// Mitsubishi GX Works2 project: REAL_PROJECT   PLC: Q03UDV

PROGRAM Manual
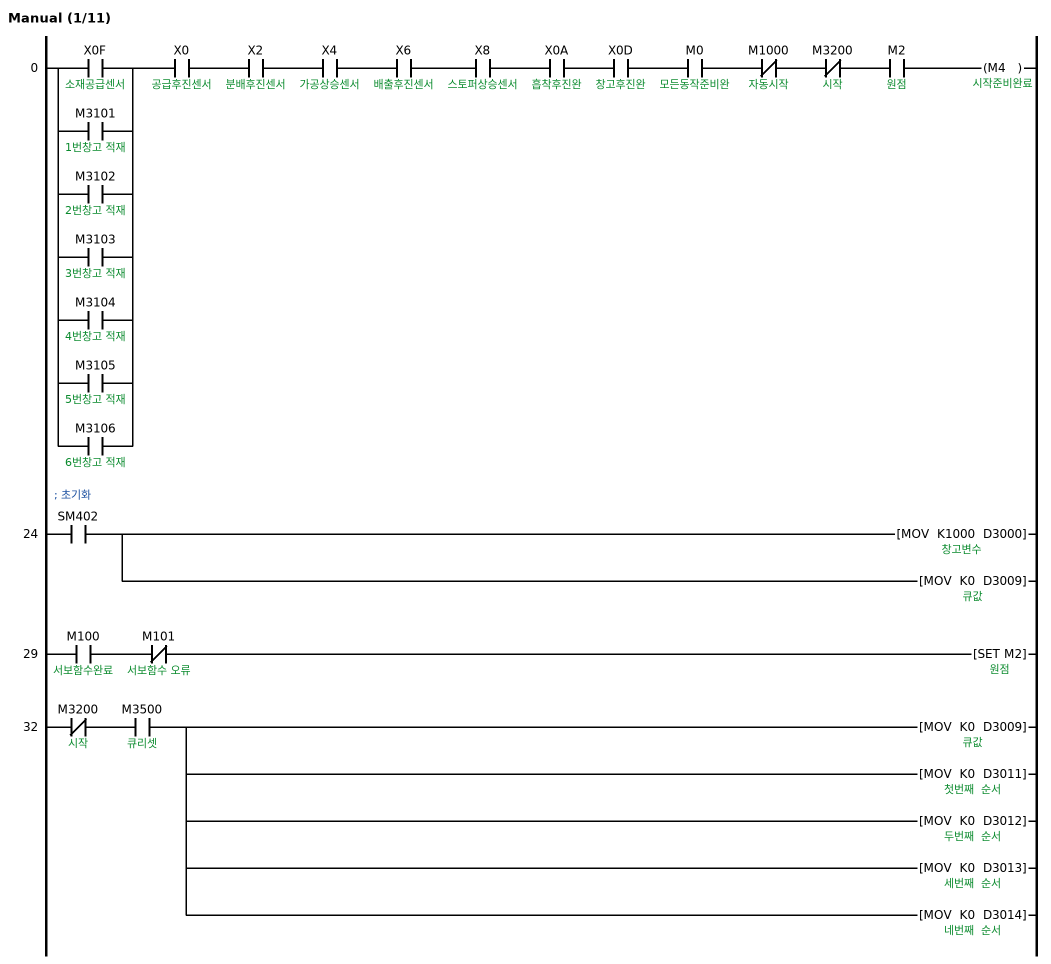
0     LD      X0F  ; 소재공급센서
      OR      M3101  ; 1번창고 적재
      OR      M3102  ; 2번창고 적재
      OR      M3103  ; 3번창고 적재
      OR      M3104  ; 4번창고 적재
      OR      M3105  ; 5번창고 적재
      OR      M3106  ; 6번창고 적재
      AND     X0  ; 공급후진센서
      AND     X2  ; 분배후진센서
      AND     X4  ; 가공상승센서
      AND     X6  ; 배출후진센서
      AND     X8  ; 스토퍼상승센서
      AND     X0A  ; 흡착후진완
      AND     X0D  ; 창고후진완
      AND     M0  ; 모든동작준비완
      ANI     M1000  ; 자동시작
      ANI     M3200  ; 시작
      AND     M2  ; 원점
      OUT     M4  ; 시작준비완료
; 초기화
24    LD      SM402
      MOV     K1000 D3000  ; 창고변수
      MOV     K0 D3009  ; 큐값
29    LD      M100  ; 서보함수완료
      ANI     M101  ; 서보함수 오류
      SET     M2  ; 원점
32    LDI     M3200  ; 시작
      AND     M3500  ; 큐리셋
      MOV     K0 D3009
      MOV     K0 D3011  ; 첫번째  순서
      MOV     K0 D3012  ; 두번째  순서
      MOV     K0 D3013  ; 세번째  순서
      MOV     K0 D3014  ; 네번째  순서
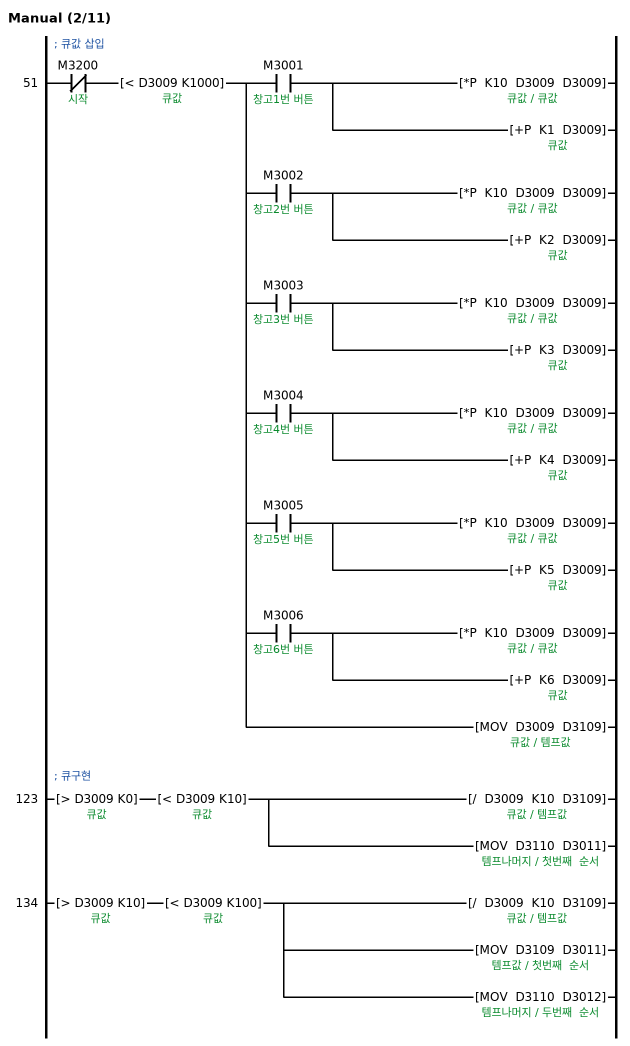
; 큐값 삽입
51    LDI     M3200  ; 시작
      AND<    D3009 K1000  ; 큐값
      MPS
      AND     M3001  ; 창고1번 버튼
      *P      K10 D3009 D3009
      +P      K1 D3009
      MRD
      AND     M3002  ; 창고2번 버튼
      *P      K10 D3009 D3009
      +P      K2 D3009
      MRD
      AND     M3003  ; 창고3번 버튼
      *P      K10 D3009 D3009
      +P      K3 D3009
      MRD
      AND     M3004  ; 창고4번 버튼
      *P      K10 D3009 D3009
      +P      K4 D3009
      MRD
      AND     M3005  ; 창고5번 버튼
      *P      K10 D3009 D3009
      +P      K5 D3009
      MRD
      AND     M3006  ; 창고6번 버튼
      *P      K10 D3009 D3009
      +P      K6 D3009
      MPP
      MOV     D3009 D3109  ; 템프값
; 큐구현
123   LD>     D3009 K0  ; 큐값
      AND<    D3009 K10  ; 큐값
      /       D3009 K10 D3109
      MOV     D3110 D3011  ; 템프나머지
134   LD>     D3009 K10  ; 큐값
      AND<    D3009 K100  ; 큐값
      /       D3009 K10 D3109
      MOV     D3109 D3011
      MOV     D3110 D3012
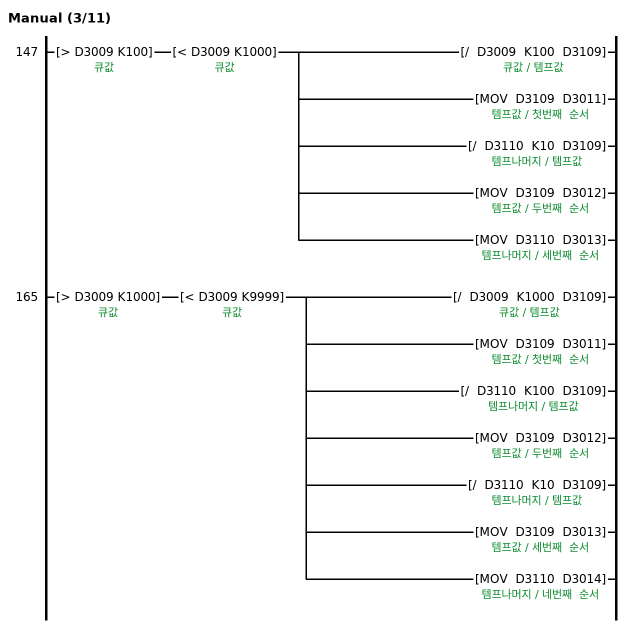
147   LD>     D3009 K100  ; 큐값
      AND<    D3009 K1000  ; 큐값
      /       D3009 K100 D3109
      MOV     D3109 D3011
      /       D3110 K10 D3109
      MOV     D3109 D3012
      MOV     D3110 D3013
165   LD>     D3009 K1000  ; 큐값
      AND<    D3009 K9999  ; 큐값
      /       D3009 K1000 D3109
      MOV     D3109 D3011
      /       D3110 K100 D3109
      MOV     D3109 D3012
      /       D3110 K10 D3109
      MOV     D3109 D3013
      MOV     D3110 D3014
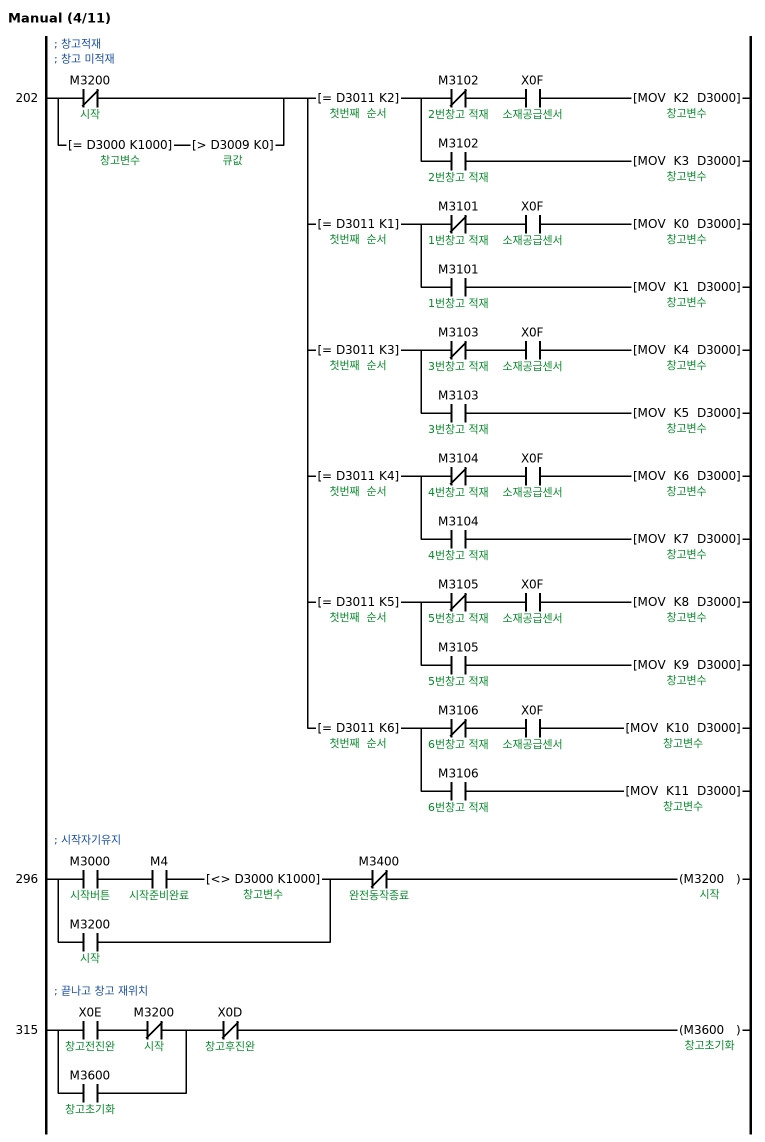
; 창고적재
; 창고 미적재
202   LDI     M3200  ; 시작
      LD=     D3000 K1000  ; 창고변수
      AND>    D3009 K0  ; 큐값
      ORB
      MPS
      AND=    D3011 K2  ; 첫번째  순서
      MPS
      ANI     M3102  ; 2번창고 적재
      AND     X0F  ; 소재공급센서
      MOV     K2 D3000
      MPP
      AND     M3102  ; 2번창고 적재
      MOV     K3 D3000
      MRD
      AND=    D3011 K1  ; 첫번째  순서
      MPS
      ANI     M3101  ; 1번창고 적재
      AND     X0F  ; 소재공급센서
      MOV     K0 D3000
      MPP
      AND     M3101  ; 1번창고 적재
      MOV     K1 D3000
      MRD
      AND=    D3011 K3  ; 첫번째  순서
      MPS
      ANI     M3103  ; 3번창고 적재
      AND     X0F  ; 소재공급센서
      MOV     K4 D3000
      MPP
      AND     M3103  ; 3번창고 적재
      MOV     K5 D3000
      MRD
      AND=    D3011 K4  ; 첫번째  순서
      MPS
      ANI     M3104  ; 4번창고 적재
      AND     X0F  ; 소재공급센서
      MOV     K6 D3000
      MPP
      AND     M3104  ; 4번창고 적재
      MOV     K7 D3000
      MRD
      AND=    D3011 K5  ; 첫번째  순서
      MPS
      ANI     M3105  ; 5번창고 적재
      AND     X0F  ; 소재공급센서
      MOV     K8 D3000
      MPP
      AND     M3105  ; 5번창고 적재
      MOV     K9 D3000
      MPP
      AND=    D3011 K6  ; 첫번째  순서
      MPS
      ANI     M3106  ; 6번창고 적재
      AND     X0F  ; 소재공급센서
      MOV     K10 D3000
      MPP
      AND     M3106  ; 6번창고 적재
      MOV     K11 D3000
; 시작자기유지
296   LD      M3000  ; 시작버튼
      AND     M4  ; 시작준비완료
      AND<>   D3000 K1000  ; 창고변수
      OR      M3200  ; 시작
      ANI     M3400  ; 완전동작종료
      OUT     M3200  ; 시작
; 끝나고 창고 재위치
315   LD      X0E  ; 창고전진완
      ANI     M3200  ; 시작
      OR      M3600  ; 창고초기화
      ANI     X0D  ; 창고후진완
      OUT     M3600  ; 창고초기화
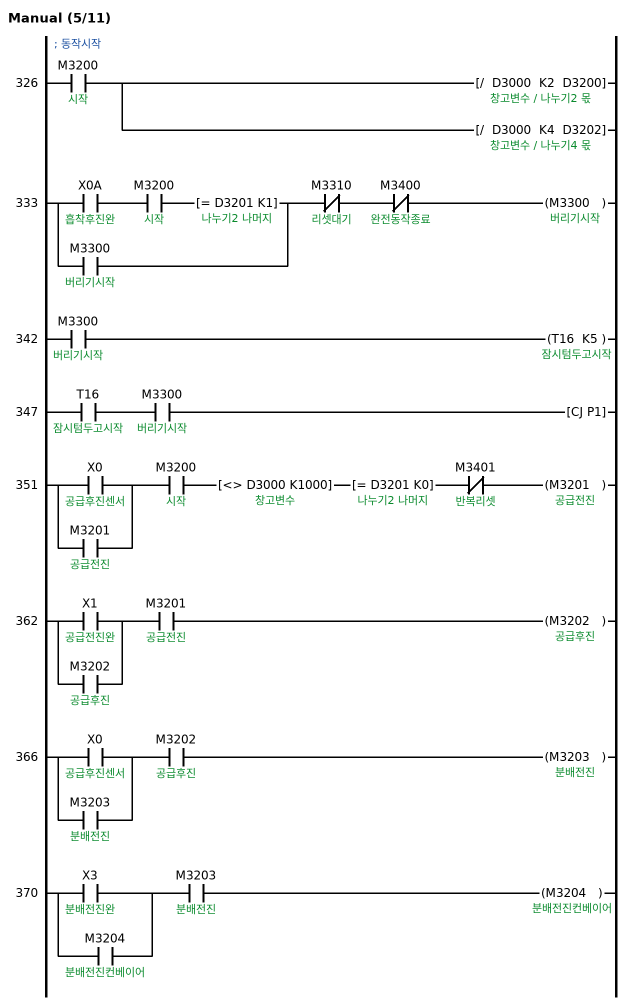
; 동작시작
326   LD      M3200  ; 시작
      /       D3000 K2 D3200  ; 나누기2 몫
      /       D3000 K4 D3202  ; 나누기4 몫
333   LD      X0A  ; 흡착후진완
      AND     M3200  ; 시작
      AND=    D3201 K1  ; 나누기2 나머지
      OR      M3300  ; 버리기시작
      ANI     M3310  ; 리셋대기
      ANI     M3400  ; 완전동작종료
      OUT     M3300  ; 버리기시작
342   LD      M3300  ; 버리기시작
      OUT     T16 K5  ; 잠시텀두고시작
347   LD      T16  ; 잠시텀두고시작
      AND     M3300  ; 버리기시작
      CJ      P1  ; 창고버리기
351   LD      X0  ; 공급후진센서
      OR      M3201  ; 공급전진
      AND     M3200  ; 시작
      AND<>   D3000 K1000  ; 창고변수
      AND=    D3201 K0  ; 나누기2 나머지
      ANI     M3401  ; 반복리셋
      OUT     M3201  ; 공급전진
362   LD      X1  ; 공급전진완
      OR      M3202  ; 공급후진
      AND     M3201  ; 공급전진
      OUT     M3202  ; 공급후진
366   LD      X0  ; 공급후진센서
      OR      M3203  ; 분배전진
      AND     M3202  ; 공급후진
      OUT     M3203  ; 분배전진
370   LD      X3  ; 분배전진완
      OR      M3204  ; 분배전진컨베이어
      AND     M3203  ; 분배전진
      OUT     M3204  ; 분배전진컨베이어
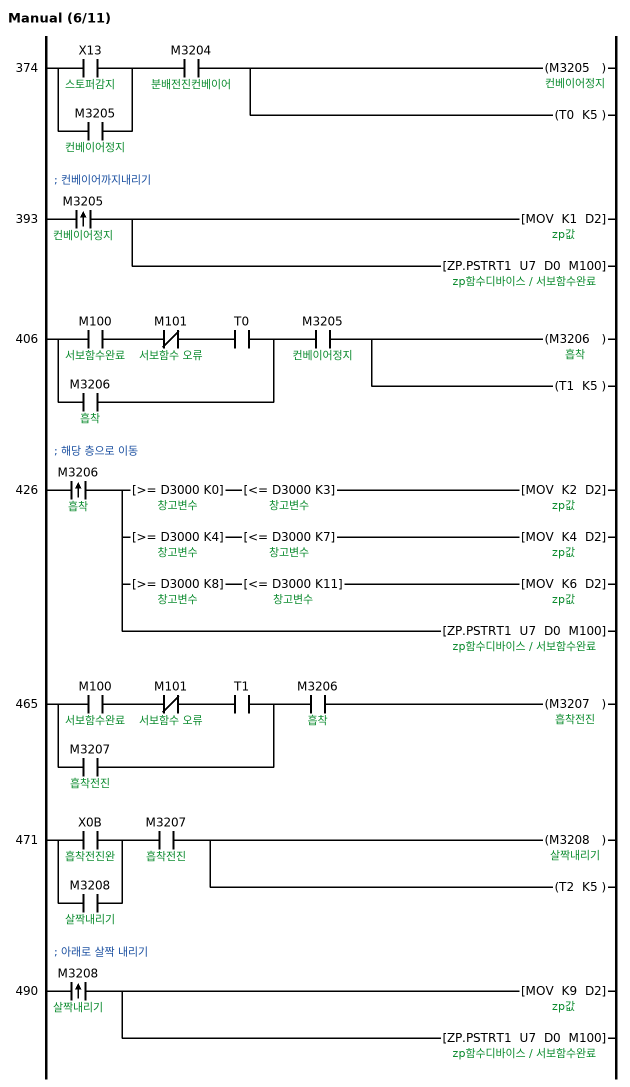
374   LD      X13  ; 스토퍼감지
      OR      M3205  ; 컨베이어정지
      AND     M3204  ; 분배전진컨베이어
      OUT     M3205  ; 컨베이어정지
      OUT     T0 K5
; 컨베이어까지내리기
393   LDP     M3205  ; 컨베이어정지
      MOV     K1 D2  ; zp값
      ZP.PSTRT1 U7 D0 M100  ; zp함수디바이스
406   LD      M100  ; 서보함수완료
      ANI     M101  ; 서보함수 오류
      AND     T0
      OR      M3206  ; 흡착
      AND     M3205  ; 컨베이어정지
      OUT     M3206  ; 흡착
      OUT     T1 K5
; 해당 층으로 이동
426   LDP     M3206  ; 흡착
      MPS
      AND>=   D3000 K0  ; 창고변수
      AND<=   D3000 K3  ; 창고변수
      MOV     K2 D2
      MRD
      AND>=   D3000 K4  ; 창고변수
      AND<=   D3000 K7  ; 창고변수
      MOV     K4 D2
      MRD
      AND>=   D3000 K8  ; 창고변수
      AND<=   D3000 K11  ; 창고변수
      MOV     K6 D2
      MPP
      ZP.PSTRT1 U7 D0 M100
465   LD      M100  ; 서보함수완료
      ANI     M101  ; 서보함수 오류
      AND     T1
      OR      M3207  ; 흡착전진
      AND     M3206  ; 흡착
      OUT     M3207  ; 흡착전진
471   LD      X0B  ; 흡착전진완
      OR      M3208  ; 살짝내리기
      AND     M3207  ; 흡착전진
      OUT     M3208  ; 살짝내리기
      OUT     T2 K5
; 아래로 살짝 내리기
490   LDP     M3208  ; 살짝내리기
      MOV     K9 D2
      ZP.PSTRT1 U7 D0 M100
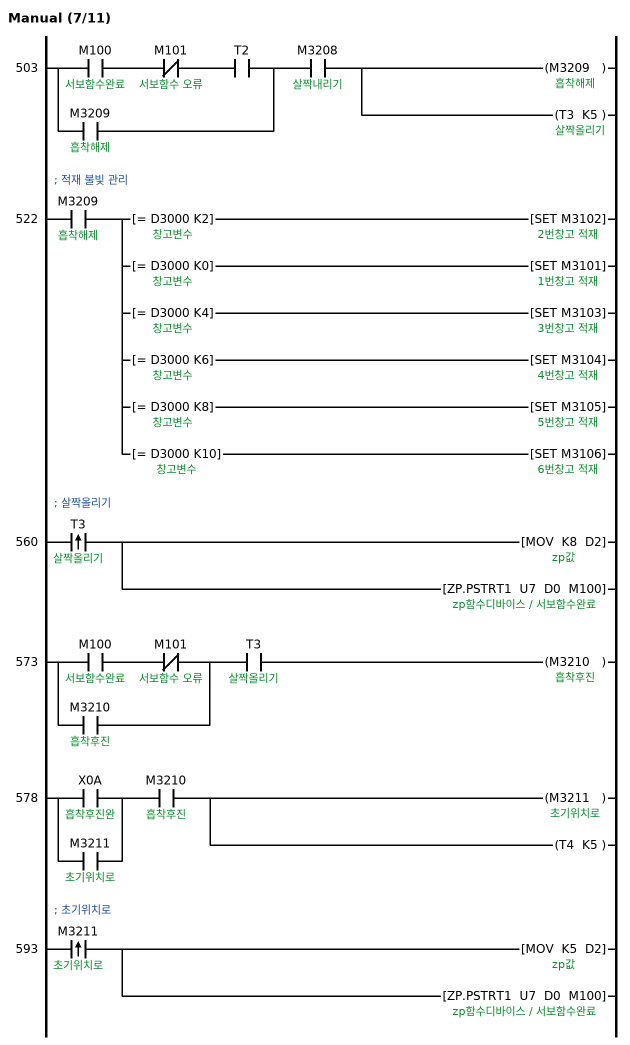
503   LD      M100  ; 서보함수완료
      ANI     M101  ; 서보함수 오류
      AND     T2
      OR      M3209  ; 흡착해제
      AND     M3208  ; 살짝내리기
      OUT     M3209  ; 흡착해제
      OUT     T3 K5  ; 살짝올리기
; 적재 불빛 관리
522   LD      M3209  ; 흡착해제
      MPS
      AND=    D3000 K2  ; 창고변수
      SET     M3102  ; 2번창고 적재
      MRD
      AND=    D3000 K0  ; 창고변수
      SET     M3101  ; 1번창고 적재
      MRD
      AND=    D3000 K4  ; 창고변수
      SET     M3103  ; 3번창고 적재
      MRD
      AND=    D3000 K6  ; 창고변수
      SET     M3104  ; 4번창고 적재
      MRD
      AND=    D3000 K8  ; 창고변수
      SET     M3105  ; 5번창고 적재
      MPP
      AND=    D3000 K10  ; 창고변수
      SET     M3106  ; 6번창고 적재
; 살짝올리기
560   LDP     T3  ; 살짝올리기
      MOV     K8 D2
      ZP.PSTRT1 U7 D0 M100
573   LD      M100  ; 서보함수완료
      ANI     M101  ; 서보함수 오류
      OR      M3210  ; 흡착후진
      AND     T3  ; 살짝올리기
      OUT     M3210  ; 흡착후진
578   LD      X0A  ; 흡착후진완
      OR      M3211  ; 초기위치로
      AND     M3210  ; 흡착후진
      OUT     M3211  ; 초기위치로
      OUT     T4 K5
; 초기위치로
593   LDP     M3211  ; 초기위치로
      MOV     K5 D2
      ZP.PSTRT1 U7 D0 M100
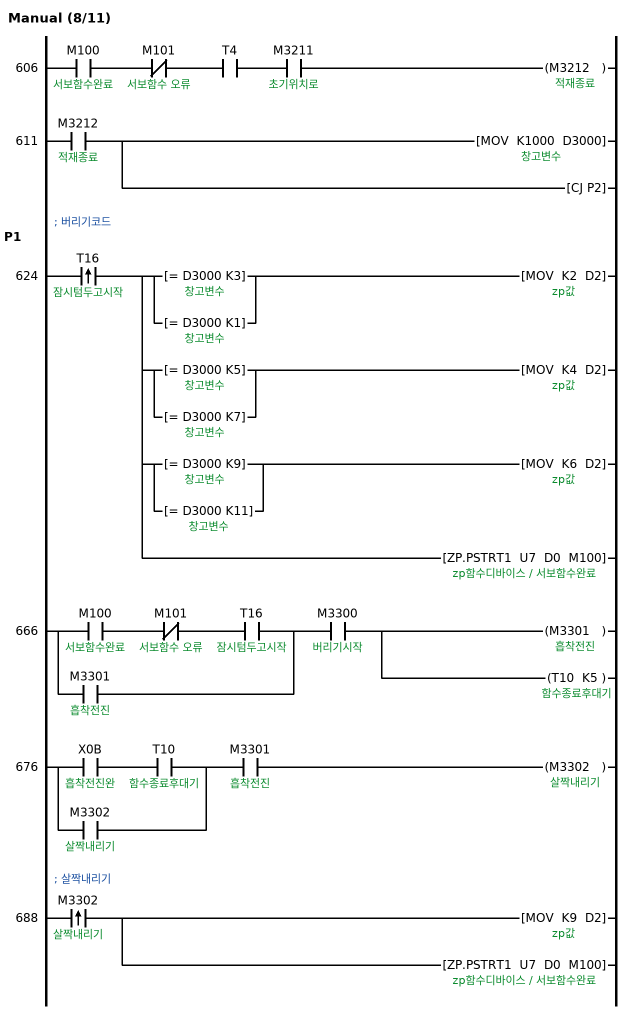
606   LD      M100  ; 서보함수완료
      ANI     M101  ; 서보함수 오류
      AND     T4
      AND     M3211  ; 초기위치로
      OUT     M3212  ; 적재종료
611   LD      M3212  ; 적재종료
      MOV     K1000 D3000
      CJ      P2  ; 버리기  로직 점프
; 버리기코드
      P1
624   LDP     T16  ; 잠시텀두고시작
      MPS
      LD=     D3000 K3  ; 창고변수
      OR=     D3000 K1  ; 창고변수
      ANB
      MOV     K2 D2
      MRD
      LD=     D3000 K5  ; 창고변수
      OR=     D3000 K7  ; 창고변수
      ANB
      MOV     K4 D2
      MRD
      LD=     D3000 K9  ; 창고변수
      OR=     D3000 K11  ; 창고변수
      ANB
      MOV     K6 D2
      MPP
      ZP.PSTRT1 U7 D0 M100
666   LD      M100  ; 서보함수완료
      ANI     M101  ; 서보함수 오류
      AND     T16  ; 잠시텀두고시작
      OR      M3301  ; 흡착전진
      AND     M3300  ; 버리기시작
      OUT     M3301  ; 흡착전진
      OUT     T10 K5  ; 함수종료후대기
676   LD      X0B  ; 흡착전진완
      AND     T10  ; 함수종료후대기
      OR      M3302  ; 살짝내리기
      AND     M3301  ; 흡착전진
      OUT     M3302  ; 살짝내리기
; 살짝내리기
688   LDP     M3302  ; 살짝내리기
      MOV     K9 D2
      ZP.PSTRT1 U7 D0 M100
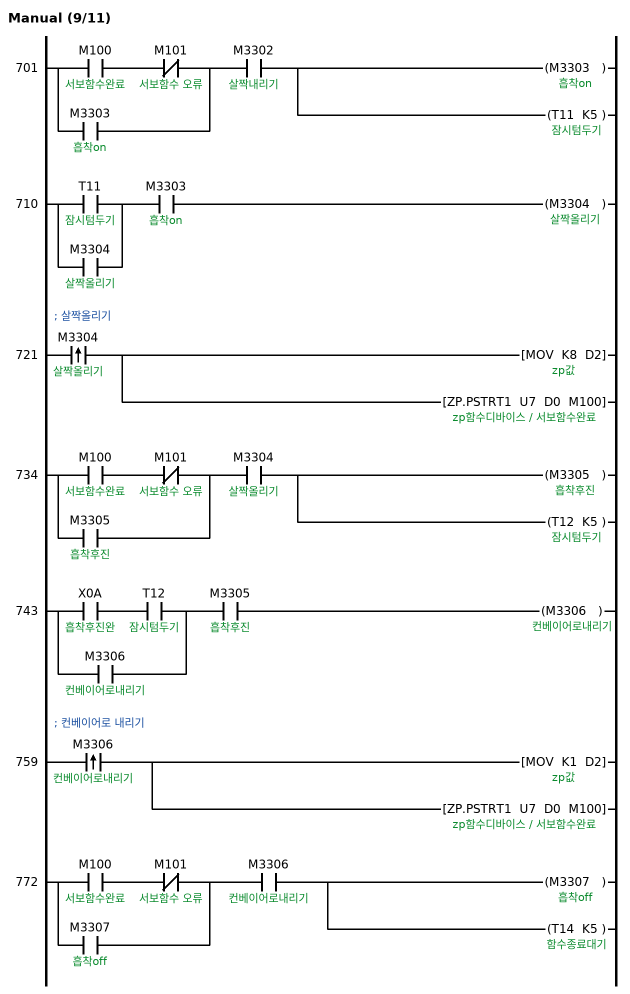
701   LD      M100  ; 서보함수완료
      ANI     M101  ; 서보함수 오류
      OR      M3303  ; 흡착on
      AND     M3302  ; 살짝내리기
      OUT     M3303  ; 흡착on
      OUT     T11 K5  ; 잠시텀두기
710   LD      T11  ; 잠시텀두기
      OR      M3304  ; 살짝올리기
      AND     M3303  ; 흡착on
      OUT     M3304  ; 살짝올리기
; 살짝올리기
721   LDP     M3304  ; 살짝올리기
      MOV     K8 D2
      ZP.PSTRT1 U7 D0 M100
734   LD      M100  ; 서보함수완료
      ANI     M101  ; 서보함수 오류
      OR      M3305  ; 흡착후진
      AND     M3304  ; 살짝올리기
      OUT     M3305  ; 흡착후진
      OUT     T12 K5  ; 잠시텀두기
743   LD      X0A  ; 흡착후진완
      AND     T12  ; 잠시텀두기
      OR      M3306  ; 컨베이어로내리기
      AND     M3305  ; 흡착후진
      OUT     M3306  ; 컨베이어로내리기
; 컨베이어로 내리기
759   LDP     M3306  ; 컨베이어로내리기
      MOV     K1 D2
      ZP.PSTRT1 U7 D0 M100
772   LD      M100  ; 서보함수완료
      ANI     M101  ; 서보함수 오류
      OR      M3307  ; 흡착off
      AND     M3306  ; 컨베이어로내리기
      OUT     M3307  ; 흡착off
      OUT     T14 K5  ; 함수종료대기
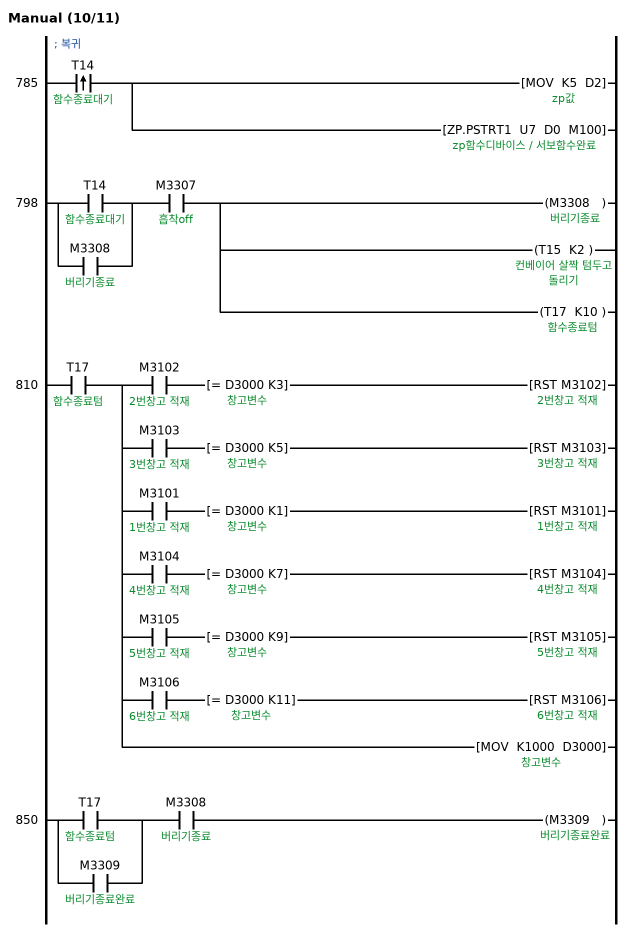
; 복귀
785   LDP     T14  ; 함수종료대기
      MOV     K5 D2
      ZP.PSTRT1 U7 D0 M100
798   LD      T14  ; 함수종료대기
      OR      M3308  ; 버리기종료
      AND     M3307  ; 흡착off
      OUT     M3308  ; 버리기종료
      OUT     T15 K2  ; 컨베이어 살짝 텀두고 돌리기
      OUT     T17 K10  ; 함수종료텀
810   LD      T17  ; 함수종료텀
      MPS
      AND     M3102  ; 2번창고 적재
      AND=    D3000 K3  ; 창고변수
      RST     M3102  ; 2번창고 적재
      MRD
      AND     M3103  ; 3번창고 적재
      AND=    D3000 K5  ; 창고변수
      RST     M3103  ; 3번창고 적재
      MRD
      AND     M3101  ; 1번창고 적재
      AND=    D3000 K1  ; 창고변수
      RST     M3101  ; 1번창고 적재
      MRD
      AND     M3104  ; 4번창고 적재
      AND=    D3000 K7  ; 창고변수
      RST     M3104  ; 4번창고 적재
      MRD
      AND     M3105  ; 5번창고 적재
      AND=    D3000 K9  ; 창고변수
      RST     M3105  ; 5번창고 적재
      MRD
      AND     M3106  ; 6번창고 적재
      AND=    D3000 K11  ; 창고변수
      RST     M3106  ; 6번창고 적재
      MPP
      MOV     K1000 D3000
850   LD      T17  ; 함수종료텀
      OR      M3309  ; 버리기종료완료
      AND     M3308  ; 버리기종료
      OUT     M3309  ; 버리기종료완료
; 큐값조정
      P2
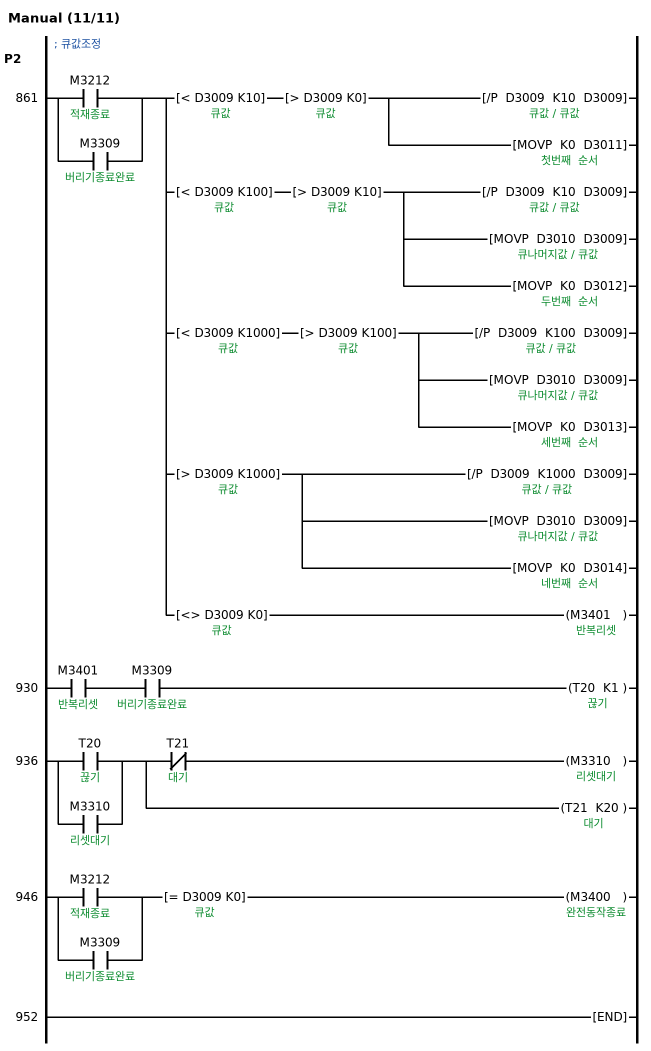
861   LD      M3212  ; 적재종료
      OR      M3309  ; 버리기종료완료
      MPS
      AND<    D3009 K10  ; 큐값
      AND>    D3009 K0  ; 큐값
      /P      D3009 K10 D3009
      MOVP    K0 D3011
      MRD
      AND<    D3009 K100  ; 큐값
      AND>    D3009 K10  ; 큐값
      /P      D3009 K10 D3009
      MOVP    D3010 D3009  ; 큐나머지값
      MOVP    K0 D3012
      MRD
      AND<    D3009 K1000  ; 큐값
      AND>    D3009 K100  ; 큐값
      /P      D3009 K100 D3009
      MOVP    D3010 D3009
      MOVP    K0 D3013
      MRD
      AND>    D3009 K1000  ; 큐값
      /P      D3009 K1000 D3009
      MOVP    D3010 D3009
      MOVP    K0 D3014
      MPP
      AND<>   D3009 K0  ; 큐값
      OUT     M3401  ; 반복리셋
930   LD      M3401  ; 반복리셋
      AND     M3309  ; 버리기종료완료
      OUT     T20 K1  ; 끊기
936   LD      T20  ; 끊기
      OR      M3310  ; 리셋대기
      MPS
      ANI     T21  ; 대기
      OUT     M3310  ; 리셋대기
      MPP
      OUT     T21 K20  ; 대기
946   LD      M3212  ; 적재종료
      OR      M3309  ; 버리기종료완료
      AND=    D3009 K0  ; 큐값
      OUT     M3400  ; 완전동작종료
952   END
END_PROGRAM

PROGRAM KeyPad
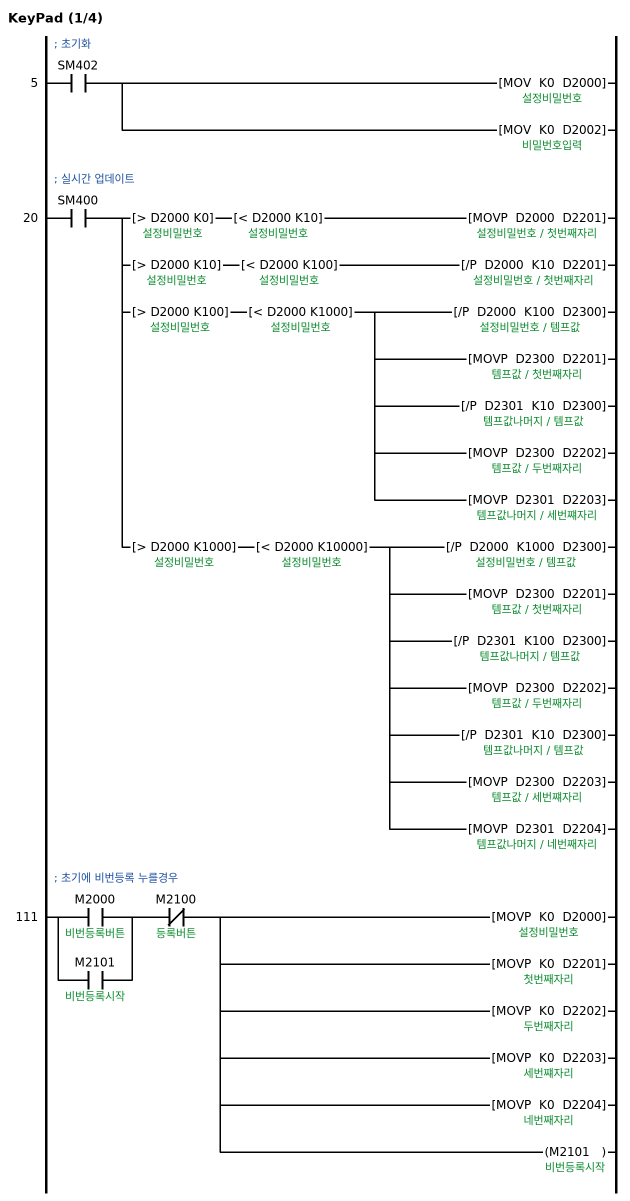
; 초기화
5     LD      SM402
      MOV     K0 D2000  ; 설정비밀번호
      MOV     K0 D2002  ; 비밀번호입력
; 실시간 업데이트
20    LD      SM400
      MPS
      AND>    D2000 K0  ; 설정비밀번호
      AND<    D2000 K10  ; 설정비밀번호
      MOVP    D2000 D2201  ; 첫번째자리
      MRD
      AND>    D2000 K10  ; 설정비밀번호
      AND<    D2000 K100  ; 설정비밀번호
      /P      D2000 K10 D2201
      MRD
      AND>    D2000 K100  ; 설정비밀번호
      AND<    D2000 K1000  ; 설정비밀번호
      /P      D2000 K100 D2300  ; 템프값
      MOVP    D2300 D2201
      /P      D2301 K10 D2300  ; 템프값나머지
      MOVP    D2300 D2202  ; 두번째자리
      MOVP    D2301 D2203  ; 세번쨰자리
      MPP
      AND>    D2000 K1000  ; 설정비밀번호
      AND<    D2000 K10000  ; 설정비밀번호
      /P      D2000 K1000 D2300
      MOVP    D2300 D2201
      /P      D2301 K100 D2300
      MOVP    D2300 D2202
      /P      D2301 K10 D2300
      MOVP    D2300 D2203
      MOVP    D2301 D2204  ; 네번째자리
; 초기에 비번등록 누를경우
111   LD      M2000  ; 비번등록버튼
      OR      M2101  ; 비번등록시작
      ANI     M2100  ; 등록버튼
      MOVP    K0 D2000
      MOVP    K0 D2201
      MOVP    K0 D2202
      MOVP    K0 D2203
      MOVP    K0 D2204
      OUT     M2101  ; 비번등록시작
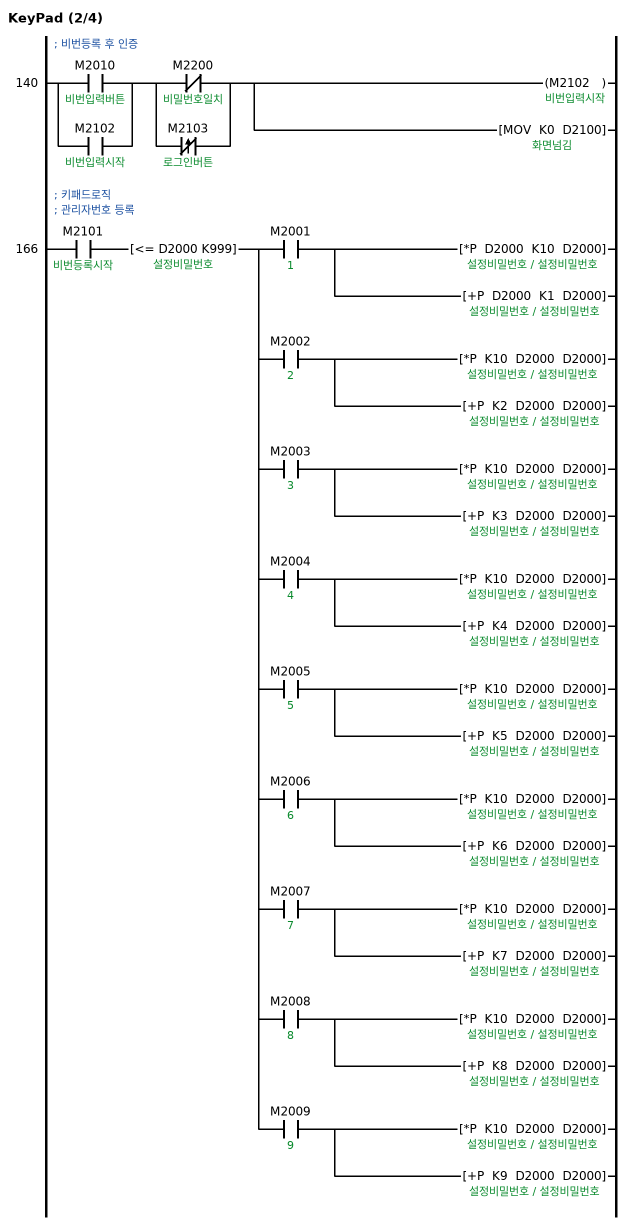
; 비번등록 후 인증
140   LD      M2010  ; 비번입력버튼
      OR      M2102  ; 비번입력시작
      LDI     M2200  ; 비밀번호일치
      ORPI    M2103  ; 로그인버튼
      ANB
      OUT     M2102  ; 비번입력시작
      MOV     K0 D2100  ; 화면넘김
; 키패드로직
; 관리자번호 등록
166   LD      M2101  ; 비번등록시작
      AND<=   D2000 K999  ; 설정비밀번호
      MPS
      AND     M2001  ; 1
      *P      D2000 K10 D2000
      +P      D2000 K1 D2000
      MRD
      AND     M2002  ; 2
      *P      K10 D2000 D2000
      +P      K2 D2000 D2000
      MRD
      AND     M2003  ; 3
      *P      K10 D2000 D2000
      +P      K3 D2000 D2000
      MRD
      AND     M2004  ; 4
      *P      K10 D2000 D2000
      +P      K4 D2000 D2000
      MRD
      AND     M2005  ; 5
      *P      K10 D2000 D2000
      +P      K5 D2000 D2000
      MRD
      AND     M2006  ; 6
      *P      K10 D2000 D2000
      +P      K6 D2000 D2000
      MRD
      AND     M2007  ; 7
      *P      K10 D2000 D2000
      +P      K7 D2000 D2000
      MRD
      AND     M2008  ; 8
      *P      K10 D2000 D2000
      +P      K8 D2000 D2000
      MPP
      AND     M2009  ; 9
      *P      K10 D2000 D2000
      +P      K9 D2000 D2000
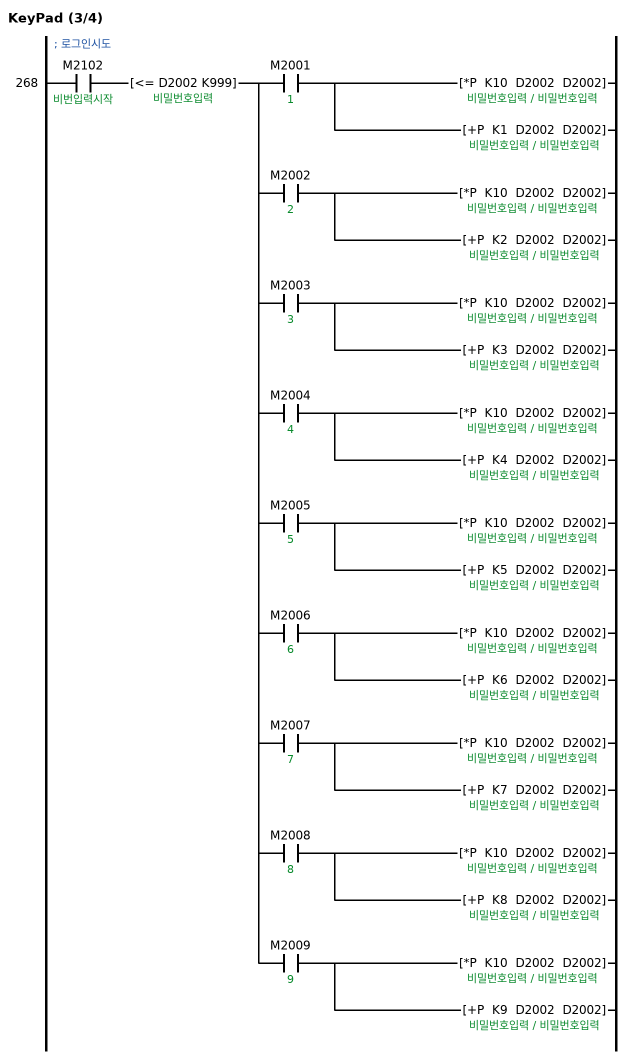
; 로그인시도
268   LD      M2102  ; 비번입력시작
      AND<=   D2002 K999  ; 비밀번호입력
      MPS
      AND     M2001  ; 1
      *P      K10 D2002 D2002
      +P      K1 D2002 D2002
      MRD
      AND     M2002  ; 2
      *P      K10 D2002 D2002
      +P      K2 D2002 D2002
      MRD
      AND     M2003  ; 3
      *P      K10 D2002 D2002
      +P      K3 D2002 D2002
      MRD
      AND     M2004  ; 4
      *P      K10 D2002 D2002
      +P      K4 D2002 D2002
      MRD
      AND     M2005  ; 5
      *P      K10 D2002 D2002
      +P      K5 D2002 D2002
      MRD
      AND     M2006  ; 6
      *P      K10 D2002 D2002
      +P      K6 D2002 D2002
      MRD
      AND     M2007  ; 7
      *P      K10 D2002 D2002
      +P      K7 D2002 D2002
      MRD
      AND     M2008  ; 8
      *P      K10 D2002 D2002
      +P      K8 D2002 D2002
      MPP
      AND     M2009  ; 9
      *P      K10 D2002 D2002
      +P      K9 D2002 D2002
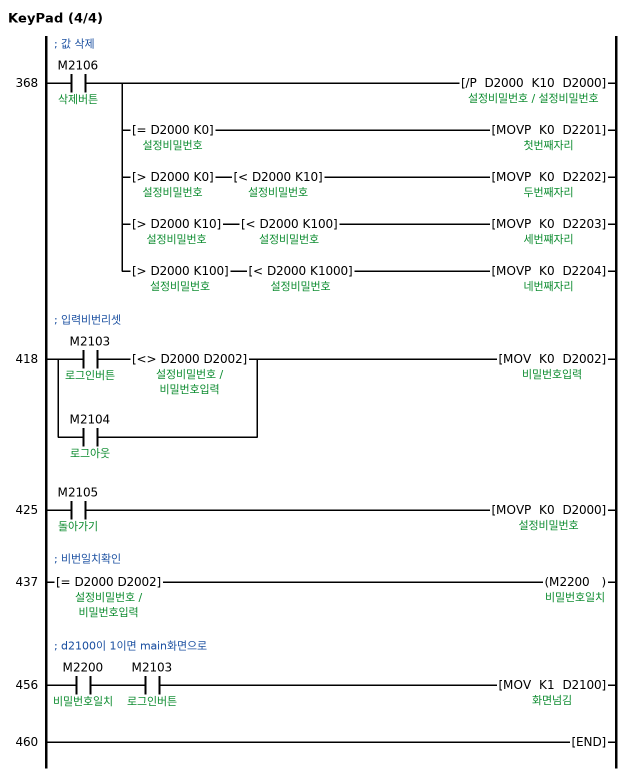
; 값 삭제
368   LD      M2106  ; 삭제버튼
      /P      D2000 K10 D2000
      MPS
      AND=    D2000 K0  ; 설정비밀번호
      MOVP    K0 D2201
      MRD
      AND>    D2000 K0  ; 설정비밀번호
      AND<    D2000 K10  ; 설정비밀번호
      MOVP    K0 D2202
      MRD
      AND>    D2000 K10  ; 설정비밀번호
      AND<    D2000 K100  ; 설정비밀번호
      MOVP    K0 D2203
      MPP
      AND>    D2000 K100  ; 설정비밀번호
      AND<    D2000 K1000  ; 설정비밀번호
      MOVP    K0 D2204
; 입력비번리셋
418   LD      M2103  ; 로그인버튼
      AND<>   D2000 D2002  ; 설정비밀번호 / 비밀번호입력
      OR      M2104  ; 로그아웃
      MOV     K0 D2002
425   LD      M2105  ; 돌아가기
      MOVP    K0 D2000
; 비번일치확인
437   LD=     D2000 D2002  ; 설정비밀번호 / 비밀번호입력
      OUT     M2200  ; 비밀번호일치
; d2100이 1이면 main화면으로
456   LD      M2200  ; 비밀번호일치
      AND     M2103  ; 로그인버튼
      MOV     K1 D2100
460   END
END_PROGRAM

PROGRAM Auto
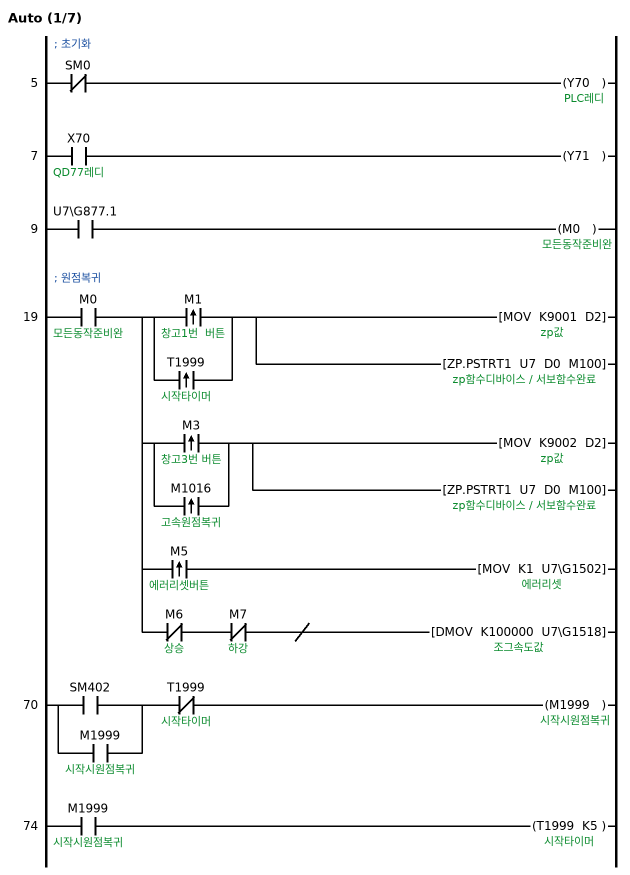
; 초기화
5     LDI     SM0
      OUT     Y70  ; PLC레디
7     LD      X70  ; QD77레디
      OUT     Y71
9     LD      U7\G877.1
      OUT     M0  ; 모든동작준비완
; 원점복귀
19    LD      M0  ; 모든동작준비완
      MPS
      LDP     M1  ; 창고1번  버튼
      ORP     T1999  ; 시작타이머
      ANB
      MOV     K9001 D2  ; zp값
      ZP.PSTRT1 U7 D0 M100  ; zp함수디바이스 / 서보함수완료
      MRD
      LDP     M3  ; 창고3번 버튼
      ORP     M1016  ; 고속원점복귀
      ANB
      MOV     K9002 D2
      ZP.PSTRT1 U7 D0 M100
      MRD
      ANDP    M5  ; 에러리셋버튼
      MOV     K1 U7\G1502  ; 에러리셋
      MPP
      ANI     M6  ; 상승
      ANI     M7  ; 하강
      INV
      DMOV    K100000 U7\G1518  ; 조그속도값
70    LD      SM402
      OR      M1999  ; 시작시원점복귀
      ANI     T1999  ; 시작타이머
      OUT     M1999  ; 시작시원점복귀
74    LD      M1999  ; 시작시원점복귀
      OUT     T1999 K5  ; 시작타이머
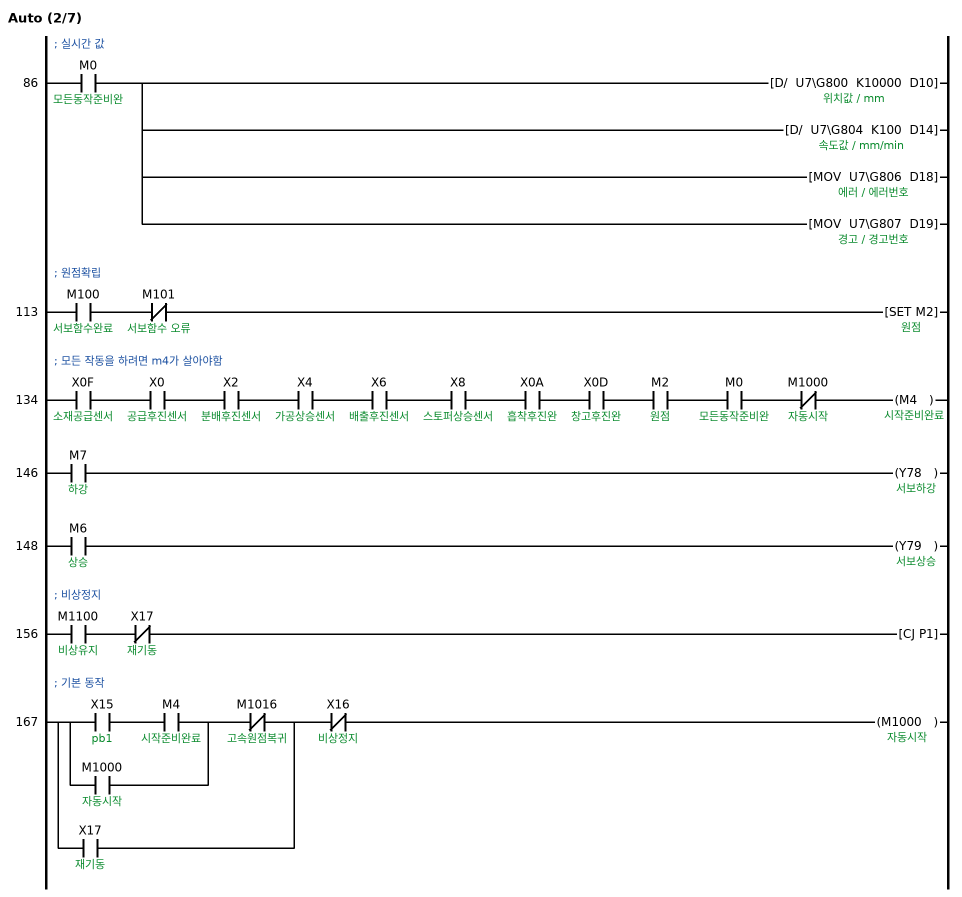
; 실시간 값
86    LD      M0  ; 모든동작준비완
      D/      U7\G800 K10000 D10  ; 위치값 / mm
      D/      U7\G804 K100 D14  ; 속도값 / mm/min
      MOV     U7\G806 D18  ; 에러 / 에러번호
      MOV     U7\G807 D19  ; 경고 / 경고번호
; 원점확립
113   LD      M100  ; 서보함수완료
      ANI     M101  ; 서보함수 오류
      SET     M2  ; 원점
; 모든 작동을 하려면 m4가 살아야함
134   LD      X0F  ; 소재공급센서
      AND     X0  ; 공급후진센서
      AND     X2  ; 분배후진센서
      AND     X4  ; 가공상승센서
      AND     X6  ; 배출후진센서
      AND     X8  ; 스토퍼상승센서
      AND     X0A  ; 흡착후진완
      AND     X0D  ; 창고후진완
      AND     M2  ; 원점
      AND     M0  ; 모든동작준비완
      ANI     M1000  ; 자동시작
      OUT     M4  ; 시작준비완료
146   LD      M7  ; 하강
      OUT     Y78  ; 서보하강
148   LD      M6  ; 상승
      OUT     Y79  ; 서보상승
; 비상정지
156   LD      M1100  ; 비상유지
      ANI     X17  ; 재기동
      CJ      P1  ; 창고버리기
; 기본 동작
167   LD      X15  ; pb1
      AND     M4  ; 시작준비완료
      OR      M1000  ; 자동시작
      ANI     M1016  ; 고속원점복귀
      OR      X17  ; 재기동
      ANI     X16  ; 비상정지
      OUT     M1000  ; 자동시작
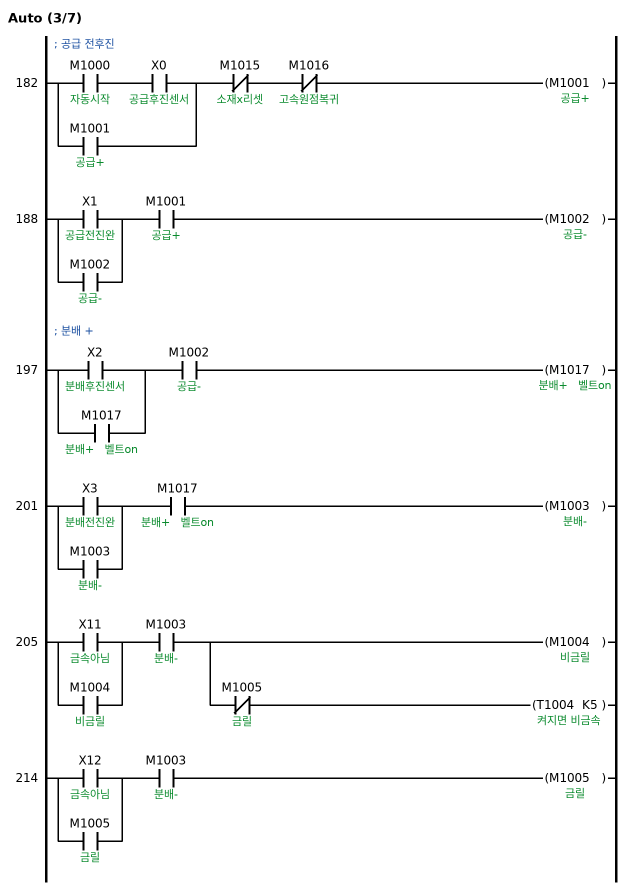
; 공급 전후진
182   LD      M1000  ; 자동시작
      AND     X0  ; 공급후진센서
      OR      M1001  ; 공급+
      ANI     M1015  ; 소재x리셋
      ANI     M1016  ; 고속원점복귀
      OUT     M1001  ; 공급+
188   LD      X1  ; 공급전진완
      OR      M1002  ; 공급-
      AND     M1001  ; 공급+
      OUT     M1002  ; 공급-
; 분배 +
197   LD      X2  ; 분배후진센서
      OR      M1017  ; 분배+   벨트on
      AND     M1002  ; 공급-
      OUT     M1017  ; 분배+   벨트on
201   LD      X3  ; 분배전진완
      OR      M1003  ; 분배-
      AND     M1017  ; 분배+   벨트on
      OUT     M1003  ; 분배-
205   LD      X11  ; 금속아님
      OR      M1004  ; 비금릴
      AND     M1003  ; 분배-
      OUT     M1004  ; 비금릴
      ANI     M1005  ; 금릴
      OUT     T1004 K5  ; 켜지면 비금속
214   LD      X12  ; 금속아님
      OR      M1005  ; 금릴
      AND     M1003  ; 분배-
      OUT     M1005  ; 금릴
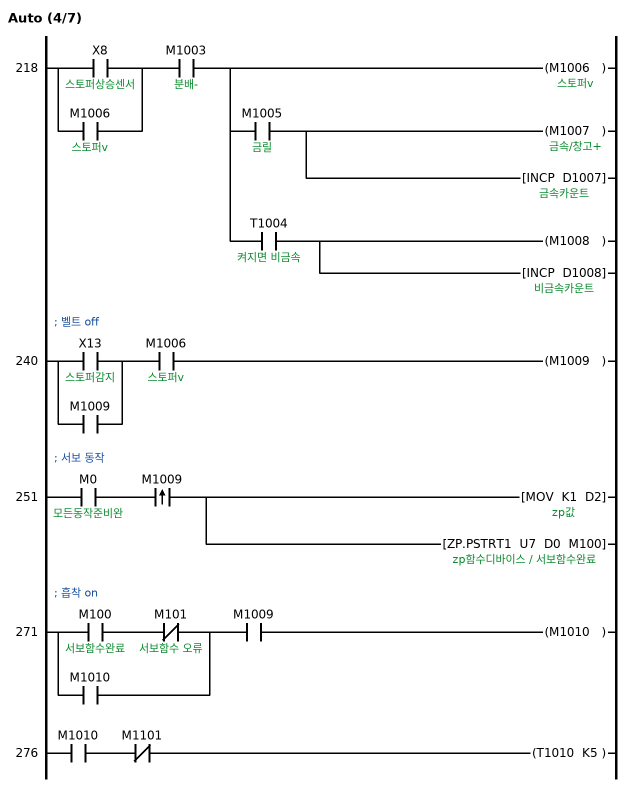
218   LD      X8  ; 스토퍼상승센서
      OR      M1006  ; 스토퍼v
      AND     M1003  ; 분배-
      OUT     M1006  ; 스토퍼v
      MPS
      AND     M1005  ; 금릴
      OUT     M1007  ; 금속/창고+
      INCP    D1007  ; 금속카운트
      MPP
      AND     T1004  ; 켜지면 비금속
      OUT     M1008
      INCP    D1008  ; 비금속카운트
; 벨트 off
240   LD      X13  ; 스토퍼감지
      OR      M1009
      AND     M1006  ; 스토퍼v
      OUT     M1009
; 서보 동작
251   LD      M0  ; 모든동작준비완
      ANDP    M1009
      MOV     K1 D2
      ZP.PSTRT1 U7 D0 M100
; 흡착 on
271   LD      M100  ; 서보함수완료
      ANI     M101  ; 서보함수 오류
      OR      M1010
      AND     M1009
      OUT     M1010
276   LD      M1010
      ANI     M1101
      OUT     T1010 K5
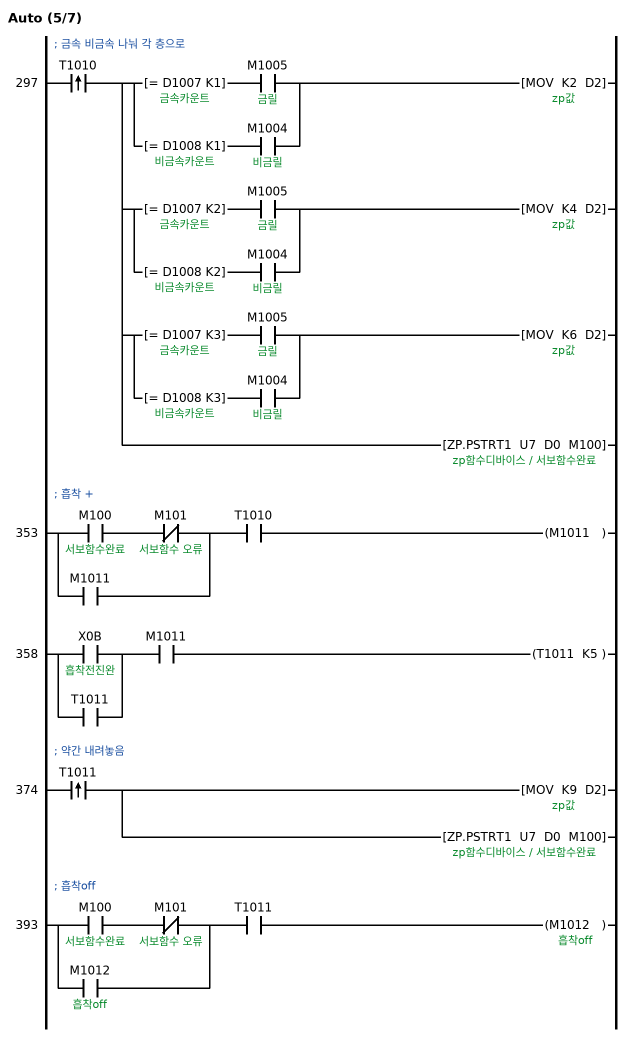
; 금속 비금속 나눠 각 층으로
297   LDP     T1010
      MPS
      LD=     D1007 K1  ; 금속카운트
      AND     M1005  ; 금릴
      LD=     D1008 K1  ; 비금속카운트
      AND     M1004  ; 비금릴
      ORB
      ANB
      MOV     K2 D2
      MRD
      LD=     D1007 K2  ; 금속카운트
      AND     M1005  ; 금릴
      LD=     D1008 K2  ; 비금속카운트
      AND     M1004  ; 비금릴
      ORB
      ANB
      MOV     K4 D2
      MRD
      LD=     D1007 K3  ; 금속카운트
      AND     M1005  ; 금릴
      LD=     D1008 K3  ; 비금속카운트
      AND     M1004  ; 비금릴
      ORB
      ANB
      MOV     K6 D2
      MPP
      ZP.PSTRT1 U7 D0 M100
; 흡착 +
353   LD      M100  ; 서보함수완료
      ANI     M101  ; 서보함수 오류
      OR      M1011
      AND     T1010
      OUT     M1011
358   LD      X0B  ; 흡착전진완
      OR      T1011
      AND     M1011
      OUT     T1011 K5
; 약간 내려놓음
374   LDP     T1011
      MOV     K9 D2
      ZP.PSTRT1 U7 D0 M100
; 흡착off
393   LD      M100  ; 서보함수완료
      ANI     M101  ; 서보함수 오류
      OR      M1012  ; 흡착off
      AND     T1011
      OUT     M1012  ; 흡착off
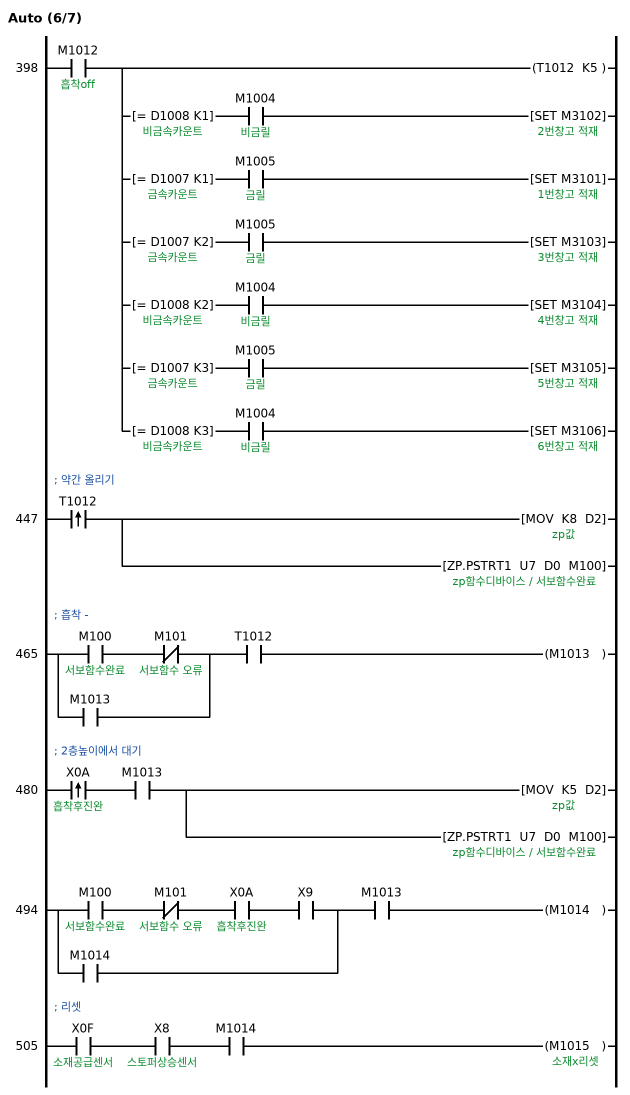
398   LD      M1012  ; 흡착off
      OUT     T1012 K5
      MPS
      AND=    D1008 K1  ; 비금속카운트
      AND     M1004  ; 비금릴
      SET     M3102  ; 2번창고 적재
      MRD
      AND=    D1007 K1  ; 금속카운트
      AND     M1005  ; 금릴
      SET     M3101  ; 1번창고 적재
      MRD
      AND=    D1007 K2  ; 금속카운트
      AND     M1005  ; 금릴
      SET     M3103  ; 3번창고 적재
      MRD
      AND=    D1008 K2  ; 비금속카운트
      AND     M1004  ; 비금릴
      SET     M3104  ; 4번창고 적재
      MRD
      AND=    D1007 K3  ; 금속카운트
      AND     M1005  ; 금릴
      SET     M3105  ; 5번창고 적재
      MPP
      AND=    D1008 K3  ; 비금속카운트
      AND     M1004  ; 비금릴
      SET     M3106  ; 6번창고 적재
; 약간 올리기
447   LDP     T1012
      MOV     K8 D2
      ZP.PSTRT1 U7 D0 M100
; 흡착 -
465   LD      M100  ; 서보함수완료
      ANI     M101  ; 서보함수 오류
      OR      M1013
      AND     T1012
      OUT     M1013
; 2층높이에서 대기
480   LDP     X0A  ; 흡착후진완
      AND     M1013
      MOV     K5 D2
      ZP.PSTRT1 U7 D0 M100
494   LD      M100  ; 서보함수완료
      ANI     M101  ; 서보함수 오류
      AND     X0A  ; 흡착후진완
      AND     X9
      OR      M1014
      AND     M1013
      OUT     M1014
; 리셋
505   LD      X0F  ; 소재공급센서
      AND     X8  ; 스토퍼상승센서
      AND     M1014
      OUT     M1015  ; 소재x리셋
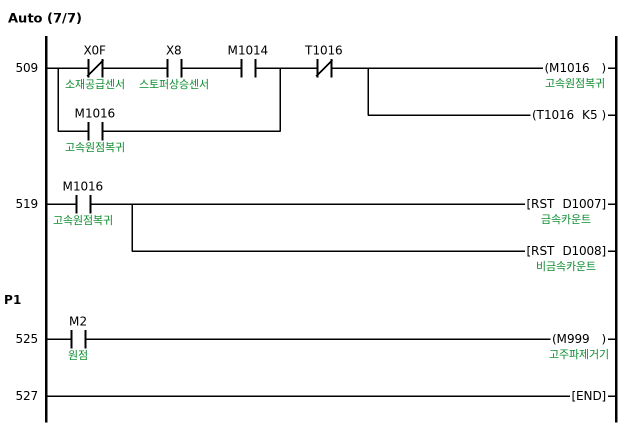
509   LDI     X0F  ; 소재공급센서
      AND     X8  ; 스토퍼상승센서
      AND     M1014
      OR      M1016  ; 고속원점복귀
      ANI     T1016
      OUT     M1016  ; 고속원점복귀
      OUT     T1016 K5
519   LD      M1016  ; 고속원점복귀
      RST     D1007  ; 금속카운트
      RST     D1008  ; 비금속카운트
      P1
525   LD      M2  ; 원점
      OUT     M999  ; 고주파제거기
527   END
END_PROGRAM

PROGRAM EMG
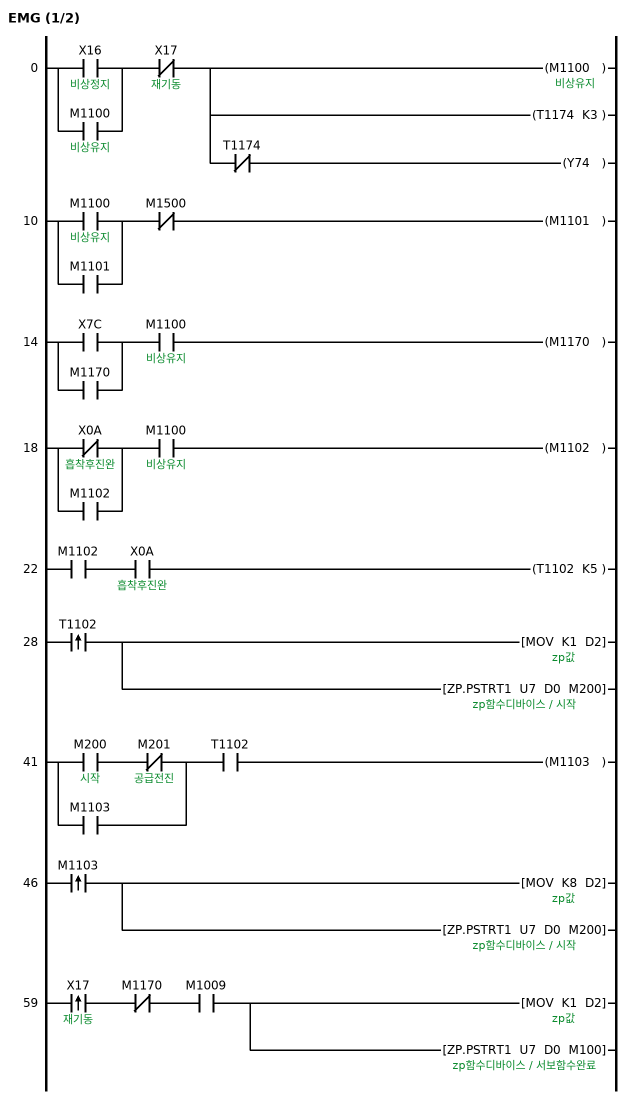
0     LD      X16  ; 비상정지
      OR      M1100  ; 비상유지
      ANI     X17  ; 재기동
      OUT     M1100  ; 비상유지
      OUT     T1174 K3
      ANI     T1174
      OUT     Y74
10    LD      M1100  ; 비상유지
      OR      M1101
      ANI     M1500
      OUT     M1101
14    LD      X7C
      OR      M1170
      AND     M1100  ; 비상유지
      OUT     M1170
18    LDI     X0A  ; 흡착후진완
      OR      M1102
      AND     M1100  ; 비상유지
      OUT     M1102
22    LD      M1102
      AND     X0A  ; 흡착후진완
      OUT     T1102 K5
28    LDP     T1102
      MOV     K1 D2  ; zp값
      ZP.PSTRT1 U7 D0 M200  ; zp함수디바이스 / 시작
41    LD      M200  ; 시작
      ANI     M201  ; 공급전진
      OR      M1103
      AND     T1102
      OUT     M1103
46    LDP     M1103
      MOV     K8 D2
      ZP.PSTRT1 U7 D0 M200
59    LDP     X17  ; 재기동
      ANI     M1170
      AND     M1009
      MOV     K1 D2
      ZP.PSTRT1 U7 D0 M100  ; 서보함수완료
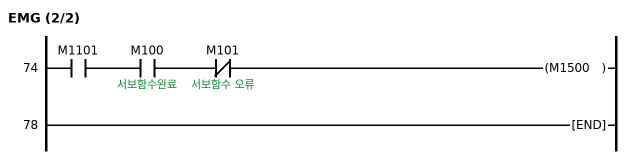
74    LD      M1101
      AND     M100  ; 서보함수완료
      ANI     M101  ; 서보함수 오류
      OUT     M1500
78    END
END_PROGRAM

PROGRAM OUTPUT
